// TIA Portal V18 export
FUNCTION_BLOCK "PIDNormal_FB_1.0"   // FB66, LAD
TITLE = Regulator PID
{ S7_Optimized_Access := 'TRUE' }
VERSION : 0.1
// stored: AutoNumber true, IsIECCheckEnabled false, IsRetainMemResEnabled false, MemoryReserve 100, SetENOAutomatically false, UDAEnableTagReadback false
   VAR_INPUT
      PV : Real := 0.0;
      ResetPID : Bool;
      SetP1 : Bool;
      SetP2 : Bool;
      SetP3 : Bool;
      SetP4 : Bool;
      SetP5 : Bool;
      ManExt : Bool;
      Scale : Bool;
   END_VAR
   VAR_OUTPUT
      Out_word : Word;
   END_VAR
   VAR_IN_OUT
      Data : "PID_DT";
   END_VAR
   VAR
      IEC_Timer_0 : IEC_TIMER;
      "Last Time" : Time := T#0ms;
      IEC_Timer_1 : IEC_TIMER;
      DeltaTimeR : Real := 0.0;
      "Always On" : Bool;
      ER : Real := 0.0;
      Last_ER : Real := 0.0;
      LMN_P : Real := 0.0;
      LMN_I : Real := 0.0;
      LMN_D : Real := 0.0;
      LMN_AUTO : Real := 0.0;
      LMN : Real;   // Wyjście regulacji 0-100%
      SP1 : Real := 1.0;   // Wartość zadana 1
      SP2 : Real;   // Wartość zadana 2
      Gain : Real := 1.2;   // Stała wzmocienia
      Ti : Time := T#2s;   // Stała czasowa Ti
      Td : Time;
      Tm_lag : Time;
      Man_ON : Bool;   // Tryb pracy: 0-automatyczny;1-manualny
      MAN : Real;   // Manualna wartość zadana
      LMN_HI : Real := 100.0;   // Maksymalne wyjście regulacji
      LMN_LO : Real := 30.0;   // Minimalne wyjście regulacji
      Reset : Bool;   // Reset układu regulacji
      ResetHMI : Bool;   // Aktualna wartość zadana
      SPAKt : Real;
      SP3 : Real;   // Wartość zadana 3
      SP4 : Real;   // Wartość zadana 4
      SP5 : Real;
   END_VAR
   VAR_TEMP
      ET : Time;
      DeltaTimeDI : DInt;
      AuxDI1 : DInt;
      AuxDI2 : DInt;
      Ti_R : Real;
      Td_R : Real;
      Tm_R : Real;
      AuxR : Real;
      AuxR2 : Real;
      DeltaER : Real;
      temp1 : Real;
      temp2 : Real;
      tempAutoMan : Bool;
      tempReset : Bool;
   END_VAR
   VAR_TEMP   // added for the SCL form of the ladder/FBD networks
      _w1 : Bool;
      _w2 : Bool;
      _w3 : Bool;
   END_VAR
BEGIN

REGION Network 1
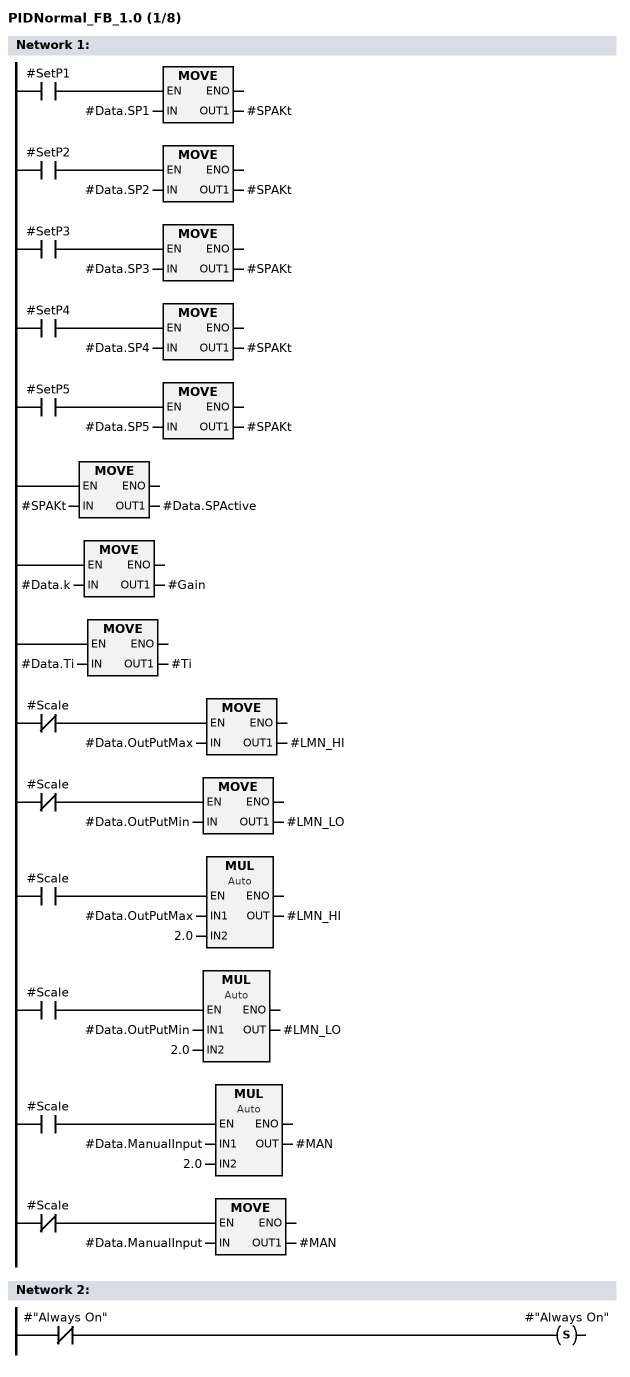
   RUNG wire#powerrail
      Contact( #SetP1 )
      { S7_GenerateENO := "TRUE" } Move(in := #Data.SP1, out1 => #SPAKt)
   END_RUNG
   RUNG wire#powerrail
      Contact( #SetP2 )
      { S7_GenerateENO := "TRUE" } Move(in := #Data.SP2, out1 => #SPAKt)
   END_RUNG
   RUNG wire#powerrail
      Contact( #SetP3 )
      { S7_GenerateENO := "TRUE" } Move(in := #Data.SP3, out1 => #SPAKt)
   END_RUNG
   RUNG wire#powerrail
      Contact( #SetP4 )
      { S7_GenerateENO := "TRUE" } Move(in := #Data.SP4, out1 => #SPAKt)
   END_RUNG
   RUNG wire#powerrail
      Contact( #SetP5 )
      { S7_GenerateENO := "TRUE" } Move(in := #Data.SP5, out1 => #SPAKt)
   END_RUNG
   RUNG wire#powerrail
      { S7_GenerateENO := "TRUE" } Move(in := #SPAKt, out1 => #Data.SPActive)
   END_RUNG
   RUNG wire#powerrail
      { S7_GenerateENO := "TRUE" } Move(in := #Data.k, out1 => #Gain)
   END_RUNG
   RUNG wire#powerrail
      { S7_GenerateENO := "TRUE" } Move(in := #Data.Ti, out1 => #Ti)
   END_RUNG
   RUNG wire#powerrail
      I_Contact( #Scale )
      { S7_GenerateENO := "TRUE" } Move(in := #Data.OutPutMax, out1 => #LMN_HI)
   END_RUNG
   RUNG wire#powerrail
      I_Contact( #Scale )
      { S7_GenerateENO := "TRUE" } Move(in := #Data.OutPutMin, out1 => #LMN_LO)
   END_RUNG
   RUNG wire#powerrail
      Contact( #Scale )
      Mul(in1 := #Data.OutPutMax, in2 := 2.0, out => #LMN_HI)
   END_RUNG
   RUNG wire#powerrail
      Contact( #Scale )
      Mul(in1 := #Data.OutPutMin, in2 := 2.0, out => #LMN_LO)
   END_RUNG
   RUNG wire#powerrail
      Contact( #Scale )
      Mul(in1 := #Data.ManualInput, in2 := 2.0, out => #MAN)
   END_RUNG
   RUNG wire#powerrail
      I_Contact( #Scale )
      { S7_GenerateENO := "TRUE" } Move(in := #Data.ManualInput, out1 => #MAN)
   END_RUNG
   // the same network as SCL:
   IF #SetP1 THEN #SPAKt := #Data.SP1; END_IF;
   IF #SetP2 THEN #SPAKt := #Data.SP2; END_IF;
   IF #SetP3 THEN #SPAKt := #Data.SP3; END_IF;
   IF #SetP4 THEN #SPAKt := #Data.SP4; END_IF;
   IF #SetP5 THEN #SPAKt := #Data.SP5; END_IF;
   #Data.SPActive := #SPAKt;
   #Gain := #Data.k;
   #Ti := #Data.Ti;
   IF NOT #Scale THEN
       #LMN_HI := #Data.OutPutMax;
       #LMN_LO := #Data.OutPutMin;
   END_IF;
   IF #Scale THEN
       #LMN_HI := #Data.OutPutMax * 2.0;
       #LMN_LO := #Data.OutPutMin * 2.0;
       #MAN := #Data.ManualInput * 2.0;
   END_IF;
   IF NOT #Scale THEN #MAN := #Data.ManualInput; END_IF;
END_REGION

REGION Network 2
   RUNG wire#powerrail
      I_Contact( #"Always On" )
      S_Coil( #"Always On" )
   END_RUNG
   // the same network as SCL:
   IF NOT #"Always On" THEN #"Always On" := TRUE; END_IF;
END_REGION

REGION Network 3
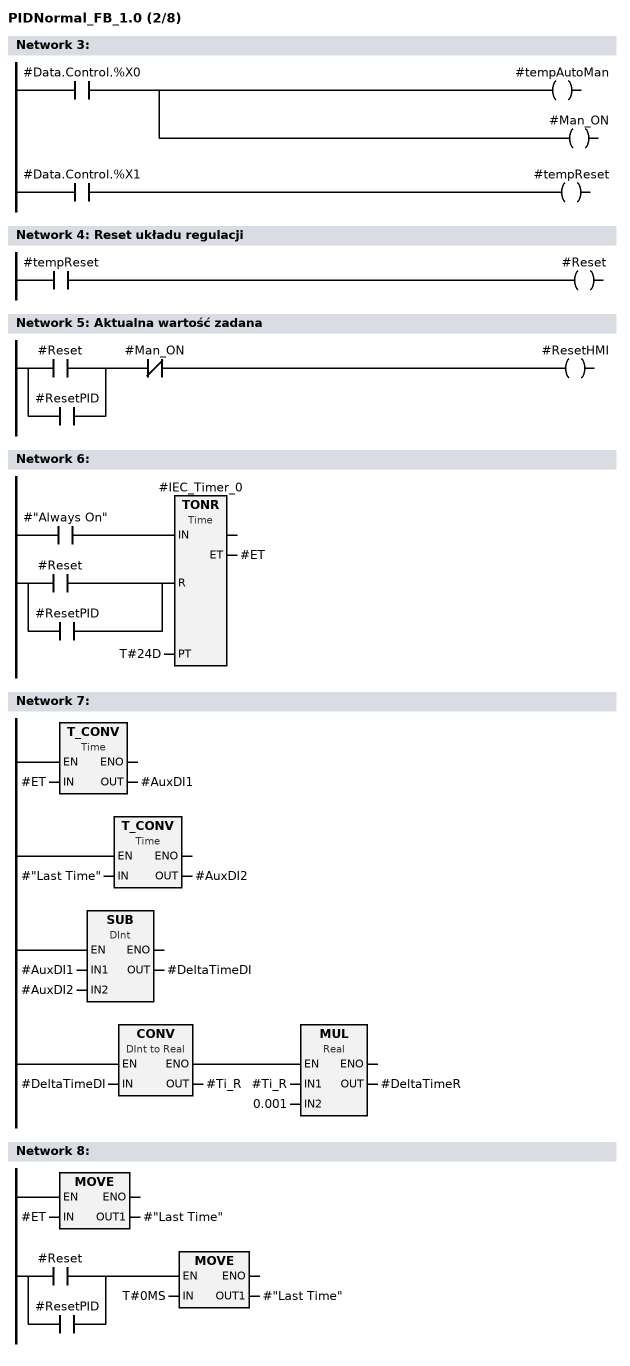
   RUNG wire#powerrail
      Contact( #Data.Control.%X0 )
      wire#w1
      Coil( #tempAutoMan )
   END_RUNG
   RUNG wire#w1
      Coil( #Man_ON )
   END_RUNG
   RUNG wire#powerrail
      Contact( #Data.Control.%X1 )
      Coil( #tempReset )
   END_RUNG
   // the same network as SCL:
   #tempAutoMan := #Data.Control.%X0;
   #Man_ON := #Data.Control.%X0;
   #tempReset := #Data.Control.%X1;
END_REGION

REGION Network 4: Reset układu regulacji
   RUNG wire#powerrail
      Contact( #tempReset )
      Coil( #Reset )
   END_RUNG
   // the same network as SCL:
   #Reset := #tempReset;
END_REGION

REGION Network 5: Aktualna wartość zadana
   RUNG wire#powerrail
      Contact( #Reset )
      wire#w1
      I_Contact( #Man_ON )
      Coil( #ResetHMI )
   END_RUNG
   RUNG wire#powerrail
      Contact( #ResetPID )
   END_RUNG wire#w1
   // the same network as SCL:
   #ResetHMI := (#Reset OR #ResetPID) AND NOT #Man_ON;
END_REGION

REGION Network 6
   RUNG wire#powerrail
      Contact( #"Always On" )
      { S7_Templates := "time_type := Time" } #IEC_Timer_0.TONR(r := wire#w1, pt := T#24D, et => #ET)
   END_RUNG
   RUNG wire#powerrail
      Contact( #Reset )
   END_RUNG wire#w1
   RUNG wire#powerrail
      Contact( #ResetPID )
   END_RUNG wire#w1
   // the same network as SCL:
   #IEC_Timer_0.TONR(IN := #"Always On", R := #Reset OR #ResetPID, PT := T#24D, ET => #ET);
END_REGION

REGION Network 7
   RUNG wire#powerrail
      { S7_Templates := "[src_type := Time, dest_type := DInt]" } T_CONV(IN := #ET, OUT => #AuxDI1)
   END_RUNG
   RUNG wire#powerrail
      { S7_Templates := "[src_type := Time, dest_type := DInt]" } T_CONV(IN := #"Last Time", OUT => #AuxDI2)
   END_RUNG
   RUNG wire#powerrail
      { S7_Templates := "SrcType := DInt"; S7_GenerateENO := "TRUE" } Sub(in1 := #AuxDI1, in2 := #AuxDI2, out => #DeltaTimeDI)
   END_RUNG
   RUNG wire#powerrail
      { S7_Templates := "[SrcType := DInt, DestType := Real]"; S7_GenerateENO := "TRUE" } Convert(in := #DeltaTimeDI, out => #Ti_R)
      { S7_Templates := "SrcType := Real"; S7_GenerateENO := "TRUE" } Mul(in1 := #Ti_R, in2 := 0.001, out => #DeltaTimeR)
   END_RUNG
   // the same network as SCL:
   // ENO of a box is taken as its EN; it also drops when the box reports an error
   T_CONV(IN := #ET, OUT => #AuxDI1);
   T_CONV(IN := #"Last Time", OUT => #AuxDI2);
   #DeltaTimeDI := #AuxDI1 - #AuxDI2;
   #Ti_R := DINT_TO_REAL(#DeltaTimeDI);
   #DeltaTimeR := #Ti_R * 0.001;
END_REGION

REGION Network 8
   RUNG wire#powerrail
      { S7_GenerateENO := "TRUE" } Move(in := #ET, out1 => #"Last Time")
   END_RUNG
   RUNG wire#powerrail
      Contact( #Reset )
      wire#w1
      { S7_GenerateENO := "TRUE" } Move(in := T#0MS, out1 => #"Last Time")
   END_RUNG
   RUNG wire#powerrail
      Contact( #ResetPID )
   END_RUNG wire#w1
   // the same network as SCL:
   #"Last Time" := #ET;
   IF #Reset OR #ResetPID THEN #"Last Time" := T#0MS; END_IF;
END_REGION

REGION Network 9
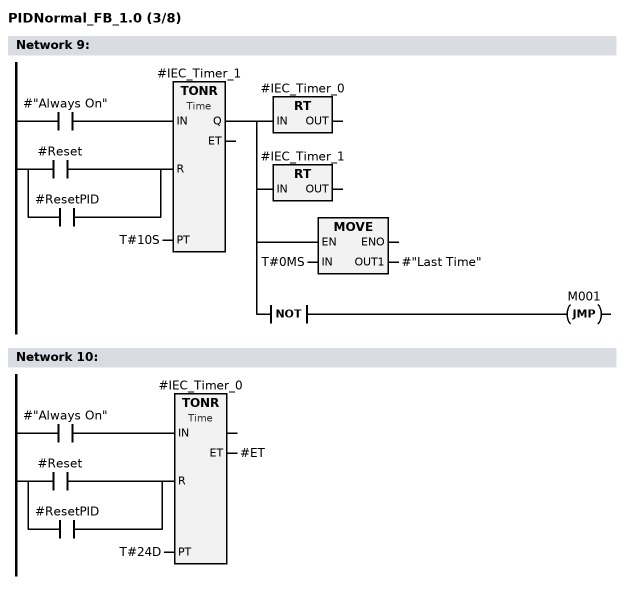
   RUNG wire#powerrail
      Contact( #"Always On" )
      { S7_Templates := "time_type := Time" } #IEC_Timer_1.TONR(r := wire#w1, pt := T#10S, et =>)
      wire#w2
      RT_Coil( #IEC_Timer_0 )
   END_RUNG
   RUNG wire#powerrail
      Contact( #Reset )
   END_RUNG wire#w1
   RUNG wire#powerrail
      Contact( #ResetPID )
   END_RUNG wire#w1
   RUNG wire#w2
      RT_Coil( #IEC_Timer_1 )
   END_RUNG
   RUNG wire#w2
      { S7_GenerateENO := "TRUE" } Move(in := T#0MS, out1 => #"Last Time")
   END_RUNG
   RUNG wire#w2
      Not()
      JumpCoil( M001 )
   END_RUNG
   // the same network as SCL:
   #IEC_Timer_1.TONR(IN := #"Always On", R := #Reset OR #ResetPID, PT := T#10S);
   IF #IEC_Timer_1.Q THEN RESET_TIMER(#IEC_Timer_0); END_IF;
   #_w1 := #IEC_Timer_1.Q;
   IF #_w1 THEN
       RESET_TIMER(#IEC_Timer_1);
       #"Last Time" := T#0MS;
   END_IF;
   IF NOT #_w1 THEN GOTO M001; END_IF;
END_REGION

REGION Network 10
   RUNG wire#powerrail
      Contact( #"Always On" )
      { S7_Templates := "time_type := Time" } #IEC_Timer_0.TONR(r := wire#w1, pt := T#24D, et => #ET)
   END_RUNG
   RUNG wire#powerrail
      Contact( #Reset )
   END_RUNG wire#w1
   RUNG wire#powerrail
      Contact( #ResetPID )
   END_RUNG wire#w1
   // the same network as SCL:
   #IEC_Timer_0.TONR(IN := #"Always On", R := #Reset OR #ResetPID, PT := T#24D, ET => #ET);
END_REGION

REGION Network 11
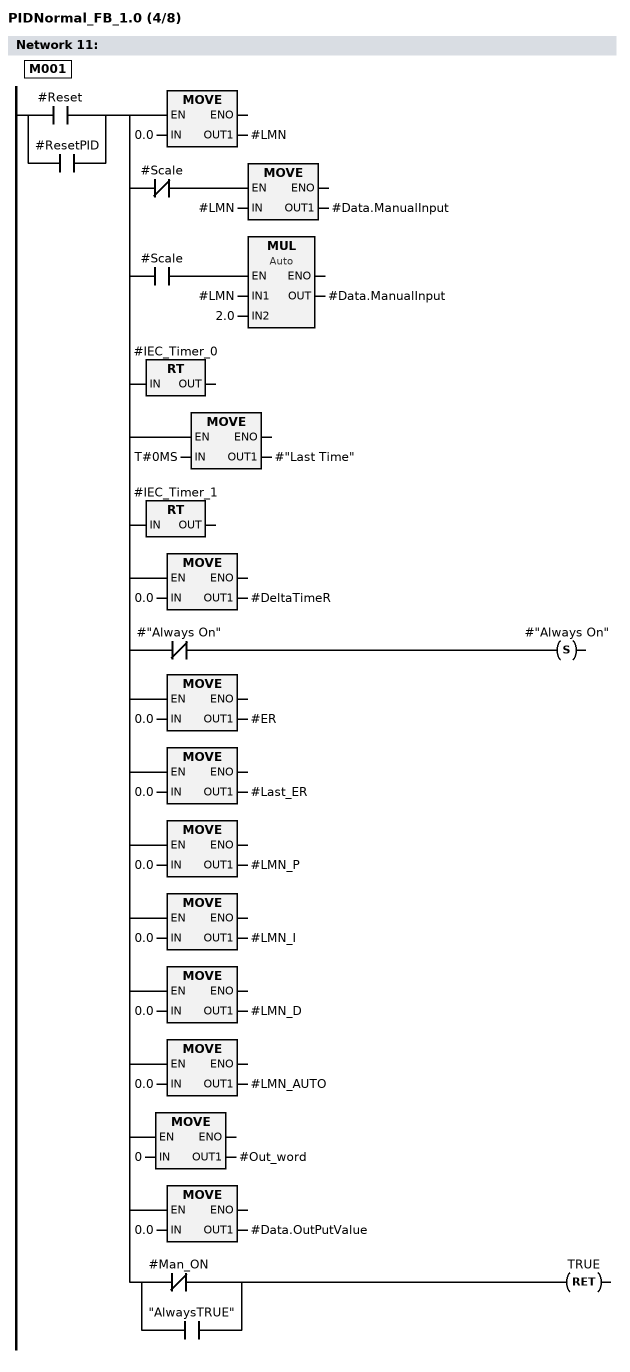
   M001:
   #_w1 := #Reset OR #ResetPID;
   IF #_w1 THEN #LMN := 0.0; END_IF;
   IF #_w1 AND NOT #Scale THEN #Data.ManualInput := #LMN; END_IF;
   IF #_w1 AND #Scale THEN #Data.ManualInput := #LMN * 2.0; END_IF;
   IF #_w1 THEN
       RESET_TIMER(#IEC_Timer_0);
       #"Last Time" := T#0MS;
       RESET_TIMER(#IEC_Timer_1);
       #DeltaTimeR := 0.0;
   END_IF;
   IF #_w1 AND NOT #"Always On" THEN #"Always On" := TRUE; END_IF;
   IF #_w1 THEN
       #ER := 0.0;
       #Last_ER := 0.0;
       #LMN_P := 0.0;
       #LMN_I := 0.0;
       #LMN_D := 0.0;
       #LMN_AUTO := 0.0;
       #Out_word := 0;
       #Data.OutPutValue := 0.0;
   END_IF;
   IF #_w1 AND (NOT #Man_ON OR "AlwaysTRUE") THEN
       ENO := TRUE;
       RETURN;
   END_IF;
END_REGION

REGION Network 12
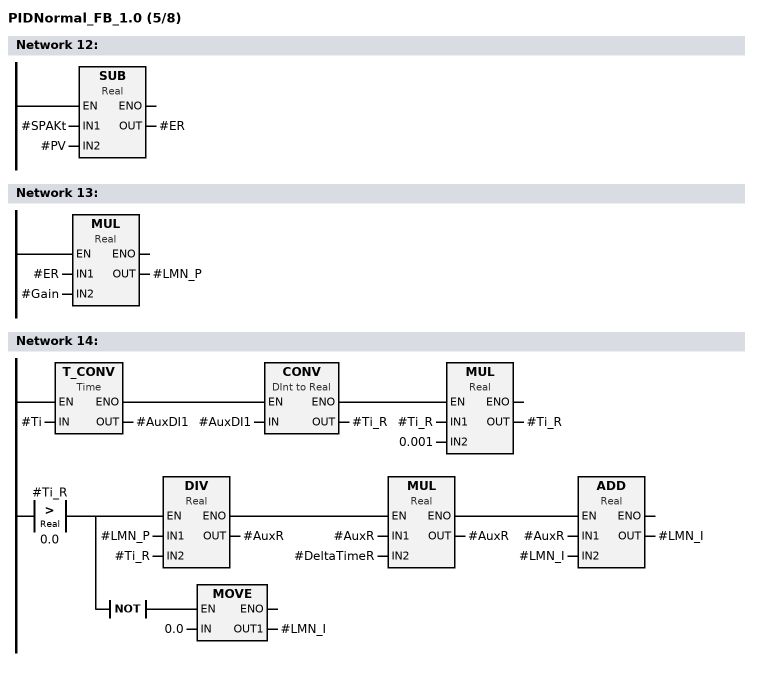
   RUNG wire#powerrail
      { S7_Templates := "SrcType := Real"; S7_GenerateENO := "TRUE" } Sub(in1 := #SPAKt, in2 := #PV, out => #ER)
   END_RUNG
   // the same network as SCL:
   #ER := #SPAKt - #PV;
END_REGION

REGION Network 13
   RUNG wire#powerrail
      { S7_Templates := "SrcType := Real"; S7_GenerateENO := "TRUE" } Mul(in1 := #ER, in2 := #Gain, out => #LMN_P)
   END_RUNG
   // the same network as SCL:
   #LMN_P := #ER * #Gain;
END_REGION

REGION Network 14
   RUNG wire#powerrail
      { S7_Templates := "[src_type := Time, dest_type := DInt]" } T_CONV(IN := #Ti, OUT => #AuxDI1)
      { S7_Templates := "[SrcType := DInt, DestType := Real]"; S7_GenerateENO := "TRUE" } Convert(in := #AuxDI1, out => #Ti_R)
      { S7_Templates := "SrcType := Real"; S7_GenerateENO := "TRUE" } Mul(in1 := #Ti_R, in2 := 0.001, out => #Ti_R)
   END_RUNG
   RUNG wire#powerrail
      { S7_Templates := "SrcType := Real" } GT_Contact(in1 := #Ti_R, in2 := 0.0)
      wire#w1
      { S7_Templates := "SrcType := Real"; S7_GenerateENO := "TRUE" } Div(in1 := #LMN_P, in2 := #Ti_R, out => #AuxR)
      { S7_Templates := "SrcType := Real"; S7_GenerateENO := "TRUE" } Mul(in1 := #AuxR, in2 := #DeltaTimeR, out => #AuxR)
      { S7_Templates := "SrcType := Real"; S7_GenerateENO := "TRUE" } Add(in1 := #AuxR, in2 := #LMN_I, out => #LMN_I)
   END_RUNG
   RUNG wire#w1
      Not()
      { S7_GenerateENO := "TRUE" } Move(in := 0.0, out1 => #LMN_I)
   END_RUNG
   // the same network as SCL:
   // ENO of a box is taken as its EN; it also drops when the box reports an error
   T_CONV(IN := #Ti, OUT => #AuxDI1, ENO => #_w1);
   IF #_w1 THEN
       #Ti_R := DINT_TO_REAL(#AuxDI1);
       #Ti_R := #Ti_R * 0.001;
   END_IF;
   #_w2 := #Ti_R > 0.0;
   IF #_w2 THEN
       #AuxR := #LMN_P / #Ti_R;
       #AuxR := #AuxR * #DeltaTimeR;
       #LMN_I := #AuxR + #LMN_I;
   END_IF;
   IF NOT #_w2 THEN #LMN_I := 0.0; END_IF;
END_REGION

REGION Network 15
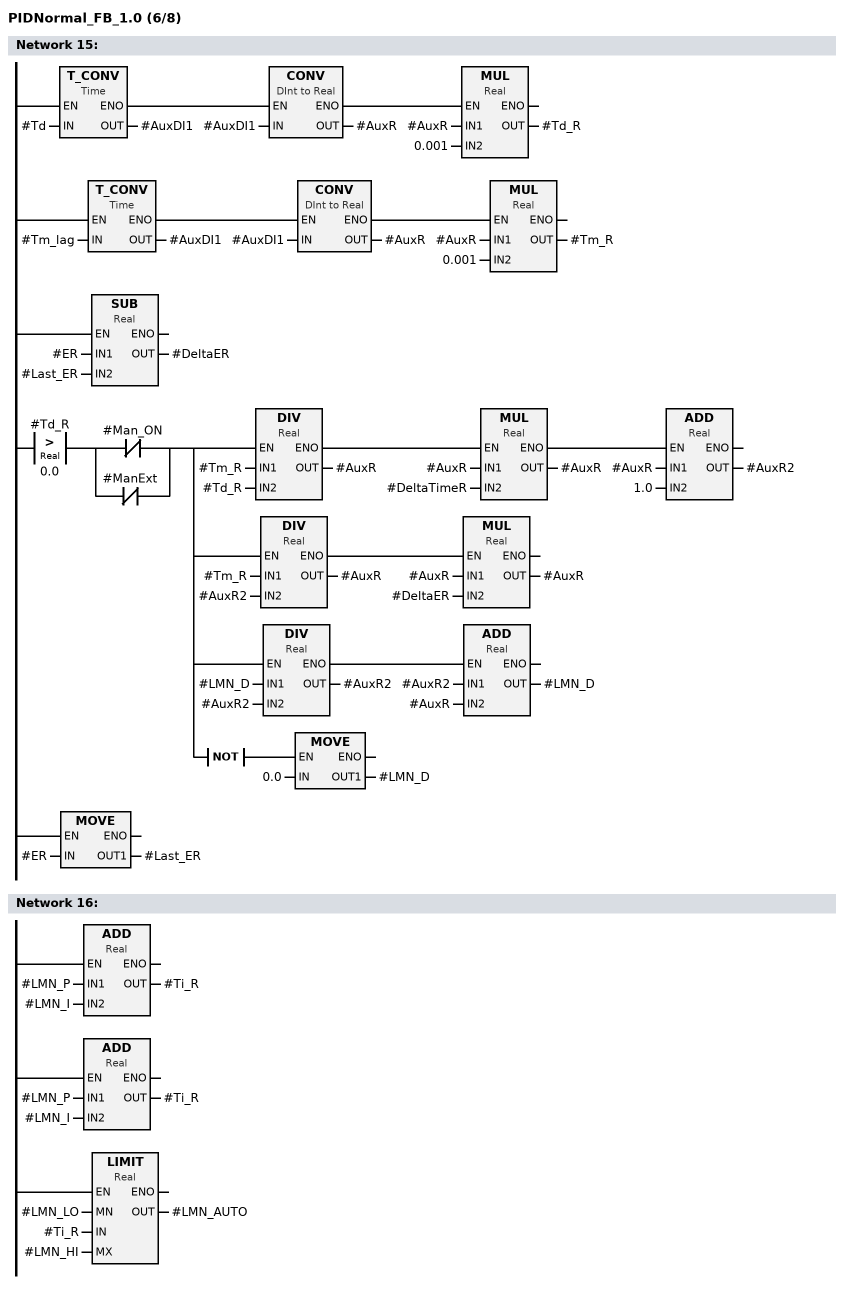
   RUNG wire#powerrail
      { S7_Templates := "[src_type := Time, dest_type := DInt]" } T_CONV(IN := #Td, OUT => #AuxDI1)
      { S7_Templates := "[SrcType := DInt, DestType := Real]"; S7_GenerateENO := "TRUE" } Convert(in := #AuxDI1, out => #AuxR)
      { S7_Templates := "SrcType := Real"; S7_GenerateENO := "TRUE" } Mul(in1 := #AuxR, in2 := 0.001, out => #Td_R)
   END_RUNG
   RUNG wire#powerrail
      { S7_Templates := "[src_type := Time, dest_type := DInt]" } T_CONV(IN := #Tm_lag, OUT => #AuxDI1)
      { S7_Templates := "[SrcType := DInt, DestType := Real]"; S7_GenerateENO := "TRUE" } Convert(in := #AuxDI1, out => #AuxR)
      { S7_Templates := "SrcType := Real"; S7_GenerateENO := "TRUE" } Mul(in1 := #AuxR, in2 := 0.001, out => #Tm_R)
   END_RUNG
   RUNG wire#powerrail
      { S7_Templates := "SrcType := Real"; S7_GenerateENO := "TRUE" } Sub(in1 := #ER, in2 := #Last_ER, out => #DeltaER)
   END_RUNG
   RUNG wire#powerrail
      { S7_Templates := "SrcType := Real" } GT_Contact(in1 := #Td_R, in2 := 0.0)
      wire#w1
      I_Contact( #Man_ON )
      wire#w2
      { S7_Templates := "SrcType := Real"; S7_GenerateENO := "TRUE" } Div(in1 := #Tm_R, in2 := #Td_R, out => #AuxR)
      { S7_Templates := "SrcType := Real"; S7_GenerateENO := "TRUE" } Mul(in1 := #AuxR, in2 := #DeltaTimeR, out => #AuxR)
      { S7_Templates := "SrcType := Real"; S7_GenerateENO := "TRUE" } Add(in1 := #AuxR, in2 := 1.0, out => #AuxR2)
   END_RUNG
   RUNG wire#w1
      I_Contact( #ManExt )
   END_RUNG wire#w2
   RUNG wire#w2
      { S7_Templates := "SrcType := Real"; S7_GenerateENO := "TRUE" } Div(in1 := #Tm_R, in2 := #AuxR2, out => #AuxR)
      { S7_Templates := "SrcType := Real"; S7_GenerateENO := "TRUE" } Mul(in1 := #AuxR, in2 := #DeltaER, out => #AuxR)
   END_RUNG
   RUNG wire#w2
      { S7_Templates := "SrcType := Real"; S7_GenerateENO := "TRUE" } Div(in1 := #LMN_D, in2 := #AuxR2, out => #AuxR2)
      { S7_Templates := "SrcType := Real"; S7_GenerateENO := "TRUE" } Add(in1 := #AuxR2, in2 := #AuxR, out => #LMN_D)
   END_RUNG
   RUNG wire#w2
      Not()
      { S7_GenerateENO := "TRUE" } Move(in := 0.0, out1 => #LMN_D)
   END_RUNG
   RUNG wire#powerrail
      { S7_GenerateENO := "TRUE" } Move(in := #ER, out1 => #Last_ER)
   END_RUNG
   // the same network as SCL:
   // ENO of a box is taken as its EN; it also drops when the box reports an error
   T_CONV(IN := #Td, OUT => #AuxDI1, ENO => #_w1);
   IF #_w1 THEN
       #AuxR := DINT_TO_REAL(#AuxDI1);
       #Td_R := #AuxR * 0.001;
   END_IF;
   T_CONV(IN := #Tm_lag, OUT => #AuxDI1, ENO => #_w2);
   IF #_w2 THEN
       #AuxR := DINT_TO_REAL(#AuxDI1);
       #Tm_R := #AuxR * 0.001;
   END_IF;
   #DeltaER := #ER - #Last_ER;
   #_w3 := (#Td_R > 0.0) AND (NOT #Man_ON OR NOT #ManExt);
   IF #_w3 THEN
       #AuxR := #Tm_R / #Td_R;
       #AuxR := #AuxR * #DeltaTimeR;
       #AuxR2 := #AuxR + 1.0;
       #AuxR := #Tm_R / #AuxR2;
       #AuxR := #AuxR * #DeltaER;
       #AuxR2 := #LMN_D / #AuxR2;
       #LMN_D := #AuxR2 + #AuxR;
   END_IF;
   IF NOT #_w3 THEN #LMN_D := 0.0; END_IF;
   #Last_ER := #ER;
END_REGION

REGION Network 16
   RUNG wire#powerrail
      { S7_Templates := "SrcType := Real"; S7_GenerateENO := "TRUE" } Add(in1 := #LMN_P, in2 := #LMN_I, out => #Ti_R)
   END_RUNG
   RUNG wire#powerrail
      { S7_Templates := "SrcType := Real"; S7_GenerateENO := "TRUE" } Add(in1 := #LMN_P, in2 := #LMN_I, out => #Ti_R)
   END_RUNG
   RUNG wire#powerrail
      { S7_Templates := "value_type := Real" } Limit(mn := #LMN_LO, in := #Ti_R, mx := #LMN_HI, out => #LMN_AUTO)
   END_RUNG
   // the same network as SCL:
   #Ti_R := #LMN_P + #LMN_I;
   #Ti_R := #LMN_P + #LMN_I;
   #LMN_AUTO := LIMIT(MN := #LMN_LO, IN := #Ti_R, MX := #LMN_HI);
END_REGION

REGION Network 17
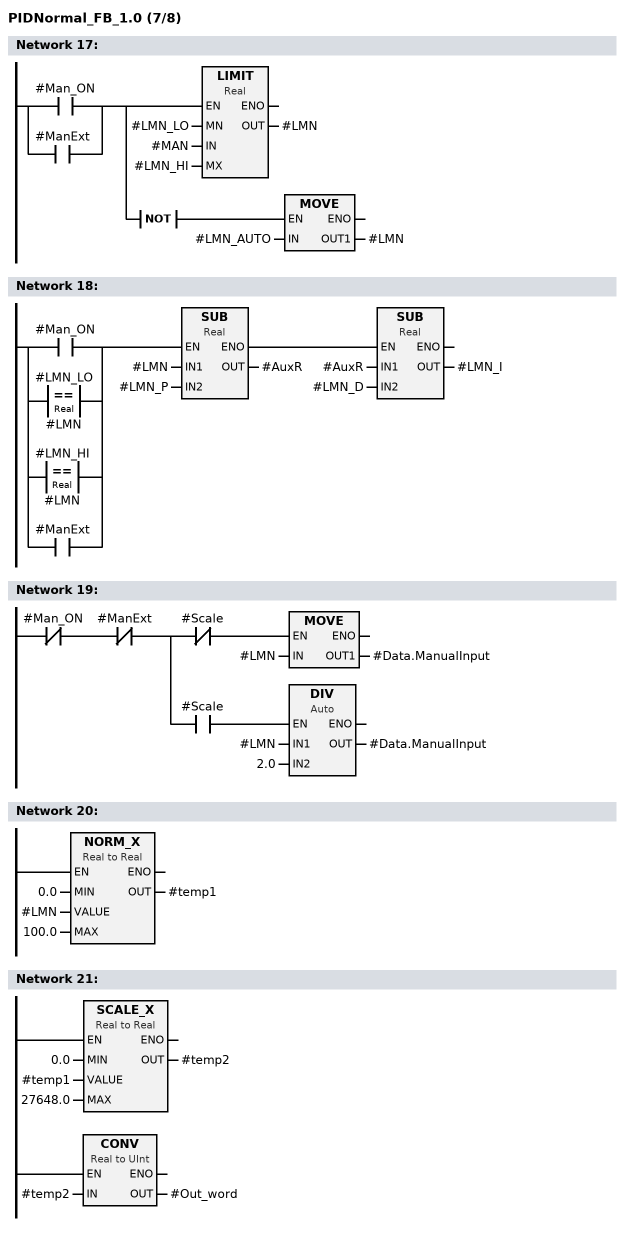
   RUNG wire#powerrail
      Contact( #Man_ON )
      wire#w1
      { S7_Templates := "value_type := Real" } Limit(mn := #LMN_LO, in := #MAN, mx := #LMN_HI, out => #LMN)
   END_RUNG
   RUNG wire#powerrail
      Contact( #ManExt )
   END_RUNG wire#w1
   RUNG wire#w1
      Not()
      { S7_GenerateENO := "TRUE" } Move(in := #LMN_AUTO, out1 => #LMN)
   END_RUNG
   // the same network as SCL:
   #_w1 := #Man_ON OR #ManExt;
   IF #_w1 THEN #LMN := LIMIT(MN := #LMN_LO, IN := #MAN, MX := #LMN_HI); END_IF;
   IF NOT #_w1 THEN #LMN := #LMN_AUTO; END_IF;
END_REGION

REGION Network 18
   RUNG wire#powerrail
      Contact( #Man_ON )
      wire#w1
      { S7_Templates := "SrcType := Real"; S7_GenerateENO := "TRUE" } Sub(in1 := #LMN, in2 := #LMN_P, out => #AuxR)
      { S7_Templates := "SrcType := Real"; S7_GenerateENO := "TRUE" } Sub(in1 := #AuxR, in2 := #LMN_D, out => #LMN_I)
   END_RUNG
   RUNG wire#powerrail
      { S7_Templates := "SrcType := Real" } EQ_Contact(in1 := #LMN_LO, in2 := #LMN)
   END_RUNG wire#w1
   RUNG wire#powerrail
      { S7_Templates := "SrcType := Real" } EQ_Contact(in1 := #LMN_HI, in2 := #LMN)
   END_RUNG wire#w1
   RUNG wire#powerrail
      Contact( #ManExt )
   END_RUNG wire#w1
   // the same network as SCL:
   // ENO of a box is taken as its EN; it also drops when the box reports an error
   IF #Man_ON OR (#LMN_LO = #LMN) OR (#LMN_HI = #LMN) OR #ManExt THEN
       #AuxR := #LMN - #LMN_P;
       #LMN_I := #AuxR - #LMN_D;
   END_IF;
END_REGION

REGION Network 19
   RUNG wire#powerrail
      I_Contact( #Man_ON )
      I_Contact( #ManExt )
      wire#w1
      I_Contact( #Scale )
      { S7_GenerateENO := "TRUE" } Move(in := #LMN, out1 => #Data.ManualInput)
   END_RUNG
   RUNG wire#w1
      Contact( #Scale )
      Div(in1 := #LMN, in2 := 2.0, out => #Data.ManualInput)
   END_RUNG
   // the same network as SCL:
   #_w1 := NOT #Man_ON AND NOT #ManExt;
   IF #_w1 AND NOT #Scale THEN #Data.ManualInput := #LMN; END_IF;
   IF #_w1 AND #Scale THEN #Data.ManualInput := #LMN / 2.0; END_IF;
END_REGION

REGION Network 20
   RUNG wire#powerrail
      { S7_Templates := "[SrcType := Real, DestType := Real]"; S7_GenerateENO := "TRUE" } Normalize(min := 0.0, value := #LMN, max := 100.0, out => #temp1)
   END_RUNG
   // the same network as SCL:
   #temp1 := NORM_X(MIN := 0.0, VALUE := #LMN, MAX := 100.0);
END_REGION

REGION Network 21
   RUNG wire#powerrail
      { S7_Templates := "[SrcType := Real, DestType := Real]"; S7_GenerateENO := "TRUE" } Scale(min := 0.0, value := #temp1, max := 27648.0, out => #temp2)
   END_RUNG
   RUNG wire#powerrail
      { S7_Templates := "[SrcType := Real, DestType := UInt]"; S7_GenerateENO := "TRUE" } Convert(in := #temp2, out => #Out_word)
   END_RUNG
   // the same network as SCL:
   #temp2 := SCALE_X(MIN := 0.0, VALUE := #temp1, MAX := 27648.0);
   #Out_word := REAL_TO_UINT(#temp2);
END_REGION

REGION Network 22
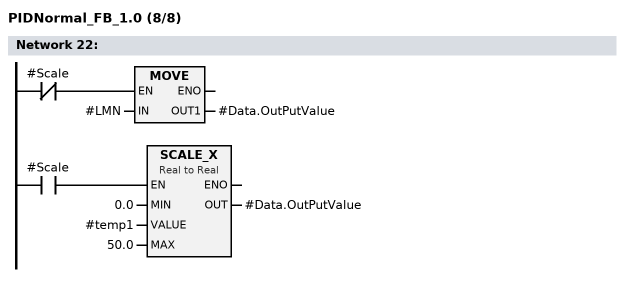
   RUNG wire#powerrail
      I_Contact( #Scale )
      { S7_GenerateENO := "TRUE" } Move(in := #LMN, out1 => #Data.OutPutValue)
   END_RUNG
   RUNG wire#powerrail
      Contact( #Scale )
      { S7_Templates := "[SrcType := Real, DestType := Real]"; S7_GenerateENO := "TRUE" } Scale(min := 0.0, value := #temp1, max := 50.0, out => #Data.OutPutValue)
   END_RUNG
   // the same network as SCL:
   IF NOT #Scale THEN #Data.OutPutValue := #LMN; END_IF;
   IF #Scale THEN #Data.OutPutValue := SCALE_X(MIN := 0.0, VALUE := #temp1, MAX := 50.0); END_IF;
END_REGION
END_FUNCTION_BLOCK
